TYPE ST_BaseEvents_RowInMemory :
STRUCT
	uiIDEvent								: UINT;				//unikalny numer zgloszenia dla całego projektu nadawany automatycznie 
	uiIDItem								: UINT;				// unikalny numer elementu w systemie
	bActive									: BOOL;
	bIgnoreRepetitions						: BOOL;				//jak true nie zliczaj powtorzeń wystapienia np komunikaty
	uiRepetitionCounter						: UINT;
	dtStart									: DT;				//poczatek wystepowania zgłoszenia
	dtFinish								: DT;				//koniec wystepowaniazgloszenia
	dtConfirmed								: DT;				// stempel potwierdzenia 
	bConfirm								: BOOL;				//informacja czy potrzebne jest potwierdzenie 
	bConfirmed								: BOOL;				//pamięta czy już potwierdzone
	eEventCategory							: E_BaseEvents_Category;
END_STRUCT
END_TYPE

(* stored: Version 1.1.0.1
   DUT ST_BaseEvents_RowInMemory: Id {29b6bf65-deca-4755-a6e5-1d76d28b8f6b} *)
